    sDescription := 'luminous efficacy';
    sUnits := 'lm W^-1';
    sCaveat := 'None';
    bFound := TRUE;
ELSIF sName = 'neutron gyromag. ratio in MHz/T' THEN
    fValue := 29.1646931; (* Units: MHz T^-1 *)
    fUncertainty := 6.9e-06;
    sDescription := 'neutron gyromag. ratio in MHz/T';
    sUnits := 'MHz T^-1';
    sCaveat := 'None';
    bFound := TRUE;
ELSIF sName = 'neutron relative atomic mass' THEN
    fValue := 1.00866491595;
    fUncertainty := 4.9e-10;
    sDescription := 'neutron relative atomic mass';
    sUnits := '';
    sCaveat := 'None';
    bFound := TRUE;
ELSIF sName = 'nuclear magneton in inverse meter per tesla' THEN
    fValue := 0.0254262341353; (* Units: m^-1 T^-1 *)
    fUncertainty := 7.8e-12;
    sDescription := 'nuclear magneton in inverse meter per tesla';
    sUnits := 'm^-1 T^-1';
    sCaveat := 'None';
    bFound := TRUE;
ELSIF sName = 'Planck constant in eV/Hz' THEN
    fValue := 4.135667696e-15; (* Units: eV Hz^-1 *)
    fUncertainty := 0;
    sDescription := 'Planck constant in eV/Hz';
    sUnits := 'eV Hz^-1';
    sCaveat := 'None';
    bFound := TRUE;
ELSIF sName = 'proton gyromag. ratio in MHz/T' THEN
    fValue := 42.577478518; (* Units: MHz T^-1 *)
    fUncertainty := 1.8e-08;
    sDescription := 'proton gyromag. ratio in MHz/T';
    sUnits := 'MHz T^-1';
    sCaveat := 'None';
    bFound := TRUE;
ELSIF sName = 'proton relative atomic mass' THEN
    fValue := 1.007276466621;
    fUncertainty := 5.3e-11;
    sDescription := 'proton relative atomic mass';
    sUnits := '';
    sCaveat := 'None';
    bFound := TRUE;
ELSIF sName = 'reduced Compton wavelength' THEN
    fValue := 3.8615926796e-13; (* Units: m *)
    fUncertainty := 1.2e-22;
    sDescription := 'reduced Compton wavelength';
    sUnits := 'm';
    sCaveat := 'None';
    bFound := TRUE;
ELSIF sName = 'reduced muon Compton wavelength' THEN
    fValue := 1.867594306e-15; (* Units: m *)
    fUncertainty := 4.2e-23;
    sDescription := 'reduced muon Compton wavelength';
    sUnits := 'm';
    sCaveat := 'None';
    bFound := TRUE;
ELSIF sName = 'reduced neutron Compton wavelength' THEN
    fValue := 2.1001941552e-16; (* Units: m *)
    fUncertainty := 1.2e-25;
    sDescription := 'reduced neutron Compton wavelength';
    sUnits := 'm';
    sCaveat := 'None';
    bFound := TRUE;
ELSIF sName = 'reduced Planck constant' THEN
    fValue := 1.054571817e-34; (* Units: J s *)
    fUncertainty := 0;
    sDescription := 'reduced Planck constant';
    sUnits := 'J s';
    sCaveat := 'None';
    bFound := TRUE;
ELSIF sName = 'reduced Planck constant in eV s' THEN
    fValue := 6.582119569e-16; (* Units: eV s *)
    fUncertainty := 0;
    sDescription := 'reduced Planck constant in eV s';
    sUnits := 'eV s';
    sCaveat := 'None';
    bFound := TRUE;
ELSIF sName = 'reduced Planck constant times c in MeV fm' THEN
    fValue := 197.3269804; (* Units: MeV fm *)
    fUncertainty := 0;
    sDescription := 'reduced Planck constant times c in MeV fm';
    sUnits := 'MeV fm';
    sCaveat := 'None';
    bFound := TRUE;
ELSIF sName = 'reduced proton Compton wavelength' THEN
    fValue := 2.10308910336e-16; (* Units: m *)
    fUncertainty := 6.4e-26;
    sDescription := 'reduced proton Compton wavelength';
    sUnits := 'm';
    sCaveat := 'None';
    bFound := TRUE;
ELSIF sName = 'reduced tau Compton wavelength' THEN
    fValue := 1.110538e-16; (* Units: m *)
    fUncertainty := 7.5e-21;
    sDescription := 'reduced tau Compton wavelength';
    sUnits := 'm';
    sCaveat := 'None';
    bFound := TRUE;
ELSIF sName = 'shielded helion gyromag. ratio in MHz/T' THEN
    fValue := 32.43409942; (* Units: MHz T^-1 *)
    fUncertainty := 3.8e-07;
    sDescription := 'shielded helion gyromag. ratio in MHz/T';
    sUnits := 'MHz T^-1';
    sCaveat := 'None';
    bFound := TRUE;
ELSIF sName = 'shielded proton gyromag. ratio in MHz/T' THEN
    fValue := 42.57638474; (* Units: MHz T^-1 *)
    fUncertainty := 4.6e-07;
    sDescription := 'shielded proton gyromag. ratio in MHz/T';
    sUnits := 'MHz T^-1';
    sCaveat := 'None';
    bFound := TRUE;
ELSIF sName = 'shielding difference of d and p in HD' THEN
    fValue := 2.02e-08;
    fUncertainty := 2e-11;
    sDescription := 'shielding difference of d and p in HD';
    sUnits := '';
    sCaveat := 'None';
    bFound := TRUE;
ELSIF sName = 'shielding difference of t and p in HT' THEN
    fValue := 2.414e-08;
    fUncertainty := 2e-11;
    sDescription := 'shielding difference of t and p in HT';
    sUnits := '';
    sCaveat := 'None';
    bFound := TRUE;
ELSIF sName = 'tau energy equivalent' THEN
    fValue := 1776.86; (* Units: MeV *)
    fUncertainty := 0.12;
    sDescription := 'tau energy equivalent';
    sUnits := 'MeV';
    sCaveat := 'None';
    bFound := TRUE;
ELSIF sName = 'triton relative atomic mass' THEN
    fValue := 3.01550071621;
    fUncertainty := 1.2e-10;
    sDescription := 'triton relative atomic mass';
    sUnits := '';
    sCaveat := 'None';
    bFound := TRUE;
ELSIF sName = 'triton to proton mag. mom. ratio' THEN
    fValue := 1.0666399191;
    fUncertainty := 2.1e-09;
    sDescription := 'triton to proton mag. mom. ratio';
    sUnits := '';
    sCaveat := 'None';
    bFound := TRUE;
ELSIF sName = 'vacuum electric permittivity' THEN
    fValue := 8.8541878128e-12; (* Units: F m^-1 *)
    fUncertainty := 1.3e-21;
    sDescription := 'vacuum electric permittivity';
    sUnits := 'F m^-1';
    sCaveat := 'None';
    bFound := TRUE;
ELSIF sName = 'vacuum mag. permeability' THEN
    fValue := 1.25663706212e-06; (* Units: N A^-2 *)
    fUncertainty := 1.9e-16;
    sDescription := 'vacuum mag. permeability';
    sUnits := 'N A^-2';
    sCaveat := 'None';
    bFound := TRUE;
ELSIF sName = 'W to Z mass ratio' THEN
    fValue := 0.88153;
    fUncertainty := 0.00017;
    sDescription := 'W to Z mass ratio';
    sUnits := '';
    sCaveat := 'None';
    bFound := TRUE;
ELSE
    bFound := FALSE;
    fValue := 0;
    fUncertainty := 0;
    sDescription := '';
    sUnits := '';
    sCaveat := '';
END_IF

END_FUNCTION_BLOCK

(* stored: Version 1.1.0.1
   POU FB_PhysicalConstants: Id {9a8d290b-fb16-1486-4e10-68afcb96fef0}, SpecialFunc None *)
